TYPE sVFD :
STRUCT
	SpeedRequested 	AT %Q* : INT;
	RunRequest		AT %Q* : UINT;
	
	CurrentSpeed 	AT %I* : INT;
	Status 			AT %I* : UINT;
END_STRUCT
END_TYPE

(* stored: Version 1.1.0.1, ProductVersion 3.1.4024.12
   DUT sVFD: Id {994e3aaf-d915-4fa7-95c1-3b8cec74d1e4} *)
